// TIA Portal V21 export
VAR_GLOBAL   // PLC tag table "KAllSensore"
END_VAR
VAR_GLOBAL CONSTANT   // user constants
   KAllSens_Spare : Int := 1;   // Spare / Scorta
   KALLSensore_02 : Int := 2;
   KALLSensore_03 : Int := 3;
   KALLSensore_04 : Int := 4;
   KALLSensore_05 : Int := 5;
   KALLSensore_06 : Int := 6;
   KALLSensore_07 : Int := 7;
   KALLSensore_08 : Int := 8;
   KALLSensore_09 : Int := 9;
   KALLSensore_10 : Int := 10;
   KALLSensore_11 : Int := 11;
   KALLSensore_12 : Int := 12;
   KALLSensore_13 : Int := 13;
   KALLSensore_14 : Int := 14;
   KALLSensore_15 : Int := 15;
   KALLSensore_16 : Int := 16;
END_VAR
